Staubli VAL3: lists_string_num.dtx

mdesc mNomSpeed
public string sString
public num nNum
